// TIA Portal V20 export
TYPE "Log_LogMsg_Header"
// stored: Namespace ProductionLine
   STRUCT
      STX : Byte;
      SOH : Byte;
      MsgLength : Int;
      MsgType : Byte;
      Reserve : Byte;
      EventLevel : Byte;
      EventGroup : Byte;
      Timestamp : Date_And_Time;
      EventID : Int;
   END_STRUCT;
END_TYPE
